FUNCTION_BLOCK FB_Ampel
VAR_INPUT
	btnReset	: BOOL;
	btnActive	: BOOL;
	bBlinktakt	: BOOL;
	config	: DUT_AmpelConfig;
END_VAR
VAR_OUTPUT
	LED_ROT	: BOOL;
	LED_GELB:	BOOL;
	LED_GRUEN: 	BOOL;
END_VAR
VAR
	state	: E_AmpelPhase := E_AmpelPhase.INIT;
	tRot	: TON;  // Leuchtdauer Rot
	tRotGelb	: TON; // Leuchtdauer RotGelb
	tGruen	: TON;		// Leuchtaduer Gruen
	tGelb	: TON;		// Leuchtdauer Gelb
END_VAR


CASE state OF
	E_AmpelPhase.INIT:
			LED_ROT	:= FALSE;
			LED_GELB := bBlinktakt;
			LED_GRUEN := FALSE;
	
	E_AmpelPhase.ROT:
			LED_ROT	:= TRUE;
			LED_GELB := FALSE;
			LED_GRUEN := FALSE;
			IF tRot.Q THEN
				state := E_AmpelPhase.ROTGELB;
			END_IF
			
	E_AmpelPhase.ROTGELB:
			LED_ROT	:= TRUE;
			LED_GELB := TRUE;
			LED_GRUEN := FALSE;
			IF tRotGelb.Q THEN
				state := E_AmpelPhase.GRUEN;
			END_IF
			
	E_AmpelPhase.GRUEN:
			LED_ROT	:= FALSE;
			LED_GELB := FALSE;
			LED_GRUEN := TRUE;
			IF tGruen.Q THEN
				state := E_AmpelPhase.GELB;
			END_IF
			
	E_AmpelPhase.GELB:
			LED_ROT	:= FALSE;
			LED_GELB := TRUE;
			LED_GRUEN := FALSE;
			IF tGelb.Q THEN
				state := E_AmpelPhase.ROT;
			END_IF
ELSE
			LED_Gelb := bBlinktakt;
			LED_ROT	:= FALSE;
			LED_GRUEN := FALSE;
END_CASE

IF btnReset THEN
	state := E_AmpelPhase.INIT;
	ELSE ;
END_IF

IF btnActive AND (state = E_AmpelPhase.INIT) THEN
	state := E_AmpelPhase.ROT;
END_IF


// Timer

tRot(	IN:=(state = E_AmpelPhase.ROT),
		PT := config.tRot);
		
tRotGelb(	IN:=(state = E_AmpelPhase.ROTGELB),
		PT := config.tRotGelb);
		
tGruen(	IN:=(state = E_AmpelPhase.GRUEN),
		PT := config.tGruen);

tGelb(	IN:=(state = E_AmpelPhase.GELB),
		PT := config.tGelb);

END_FUNCTION_BLOCK

(* stored: Version 1.1.0.1, ProductVersion 3.1.4024.12
   POU FB_Ampel: Id {aaddba8e-ced5-4396-9c8c-6bc2ed214f5f}, SpecialFunc None *)
